// TIA Portal V17 export
// export: Created 2026-04-13T11:12:45.2321993Z, ExportSetting WithDefaults, DisplayName Totally Integrated Automation Portal, DisplayVersion V17 Update 4, DisplayName TIA Portal Openness, DisplayVersion V17 Update 4, DisplayName TIA Portal Version Control Interface, DisplayVersion V17, DisplayName SINAMICS Startdrive Advanced, DisplayVersion V17, DisplayName SINAMICS Startdrive G130, G150, S120, S150, SINAMICS MV, S210, DisplayVersion V17, DisplayName SINAMICS Startdrive G110M, G120, G120C, G120D, G120P, G115D, DisplayVersion V17, DisplayName STEP 7 Professional, DisplayVersion V17 Update 4, DisplayName STEP 7 Safety, DisplayVersion V17, DisplayName WinCC Professional, DisplayVersion V17 Update 4
VAR_GLOBAL   // PLC tag table "COM"
   CSJ时间更改 AT %M50.2 : Bool;
   CBD本地读 AT %MW54 : Int;
   CJF进温SW写 AT %MW56 : Int;
   CJB搅拌1温SW写 AT %MW58 : Int;
   CJB搅拌2温SW写 AT %MW60 : Int;
END_VAR
